PROGRAM RobotMapping
VAR
	TmpByte : BYTE;
	DelayRobOffOutput : TON := (PT:=T#5S);
	TOutCom : TOF := (PT:=T#1S);
	RobotOff : BOOL := FALSE;
END_VAR

//--- If EIP communication is running -----------------
TOutCom(IN :=(GVL_Robot_Io_Map.uintD4_B17_EIB_constate = 0));

//update outputs
IF (TOutCom.Q) THEN
//--- Power Cabinet Outputs from Robot--------------------------------
	//EL2008 (T3)
	GVL_Robot_Io_Map.bOutT3_PLC 		:= GVL_Robot_Io_Map.bInT3_EIP;
	
	DelayRobOffOutput(IN := FALSE);
ELSE //--- Else write 0 to outputs
	GVL_Robot_Io_Map.bOutT3_PLC 		:= 0;
	DelayRobOffOutput(IN := TRUE);
END_IF

//--- Power Cabinet Inputs to Robot --------------------------------
	//EL1008 (T2)
GVL_Robot_Io_Map.bOutT2_EIP 		:= GVL_Robot_Io_Map.bInT2_PLC ;

END_PROGRAM

(* stored: Version 1.1.0.1, ProductVersion 3.1.4024.9
   POU RobotMapping: Id {90c0f3eb-dfba-4bfe-8818-505db9a89bcc}, SpecialFunc None *)
